(* Logix 5000 project; controller VET 1756-L62 rev 19.52; software revision 19.01; part 26 of 27 *)
(* tags used below, declared in another part *)
   _Sel_Comun : Selector;   // Comun selectores
   _Sel_eqp : Sel_eqp[300];   // Equipos Select
   _Sel_eqp_comun : Sel_eqp;   // Comun equqipos selector
   _Selector : Selector[80];
   Aux : DINT[40];
   Borrar : DINT[100];
   Color_aux : INT[1000];
   ecfgcom : Eqp_Cfg;
   eqpcom : Equipo;   // Comun Equipos
   OrigCom2 : Origen;
   SetDInt : DINT[500];
   Table1 : DINT[100];
   ti : Index;
   _BatCode : DINT[100];
   _Codes : DINT[500];
   _Eqp : Equipo[800];
   _Eqp_Cfg : Eqp_Cfg[800];
   _Origen : Origen[40];
   _Typlgie : Eqp_Typologie[800];   // Process Flow Typologie
   automat : DINT[100];
   comandos : DINT[10];
   DRT : DRTs[10];
   Set_Global : DINT[20];
   Tab_ODS : Tab_O_D_Orig;   // Tabla Origen Destino
(* Typlgie, continued *)

ROUTINE Main   (* ladder *)
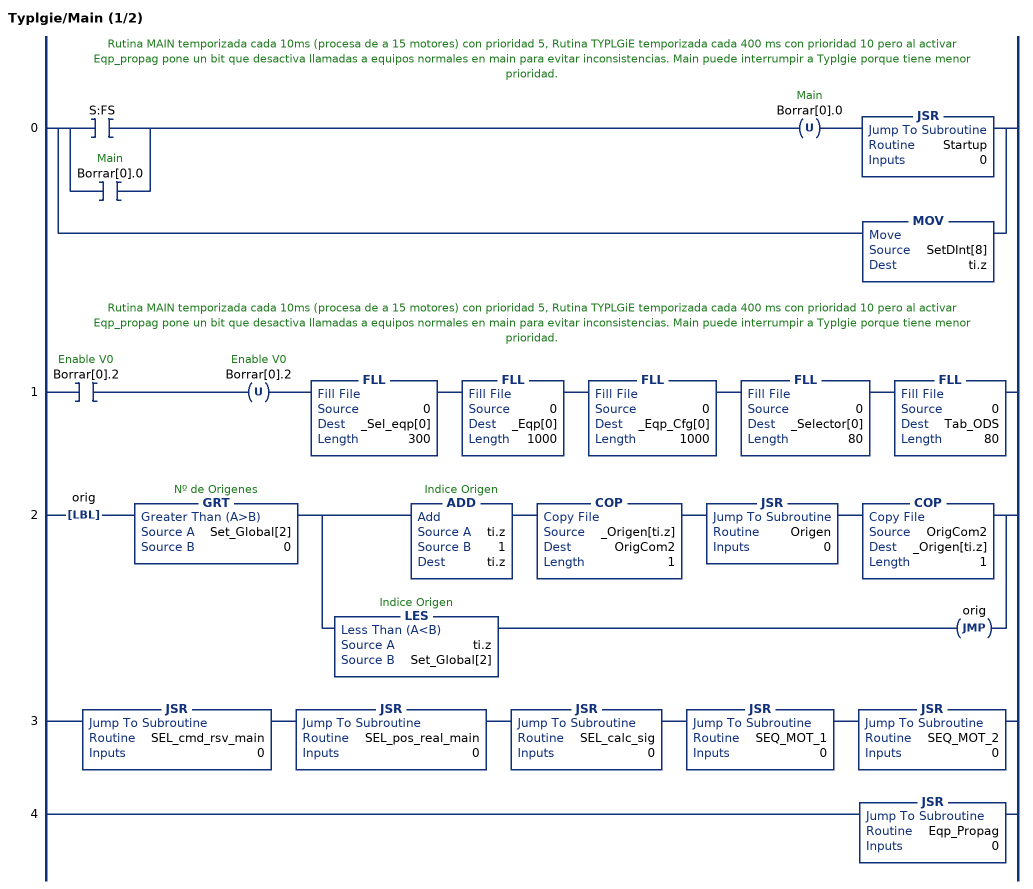
   // Rutina MAIN temporizada cada 10ms (procesa de a 15 motores) con prioridad 5, Rutina TYPLGiE temporizada cada 400 ms con prioridad 10 pero al activar Eqp_propag pone un bit que desactiva llamadas a equipos normales en main para evitar inconsistencias. Main puede interrumpir a Typlgie porque tiene menor prioridad.
   0: [[XIC(S:FS) ,XIC(Borrar[0].0) ] OTU(Borrar[0].0) JSR(Startup,0) ,MOV(SetDInt[8],ti.z) ];
   // Rutina MAIN temporizada cada 10ms (procesa de a 15 motores) con prioridad 5, Rutina TYPLGiE temporizada cada 400 ms con prioridad 10 pero al activar Eqp_propag pone un bit que desactiva llamadas a equipos normales en main para evitar inconsistencias. Main puede interrumpir a Typlgie porque tiene menor prioridad.
   1: XIC(Borrar[0].2)OTU(Borrar[0].2)FLL(0,_Sel_eqp[0],300)FLL(0,_Eqp[0],1000)FLL(0,_Eqp_Cfg[0],1000)FLL(0,_Selector[0],80)FLL(0,Tab_ODS,80);
   2: LBL(orig)GRT(Set_Global[2],0)[ADD(ti.z,1,ti.z) COP(_Origen[ti.z],OrigCom2,1) JSR(Origen,0) COP(OrigCom2,_Origen[ti.z],1) ,LES(ti.z,Set_Global[2]) JMP(orig) ];
   3: JSR(SEL_cmd_rsv_main,0)JSR(SEL_pos_real_main,0)JSR(SEL_calc_sig,0)JSR(SEQ_MOT_1,0)JSR(SEQ_MOT_2,0);
   4: JSR(Eqp_Propag,0);
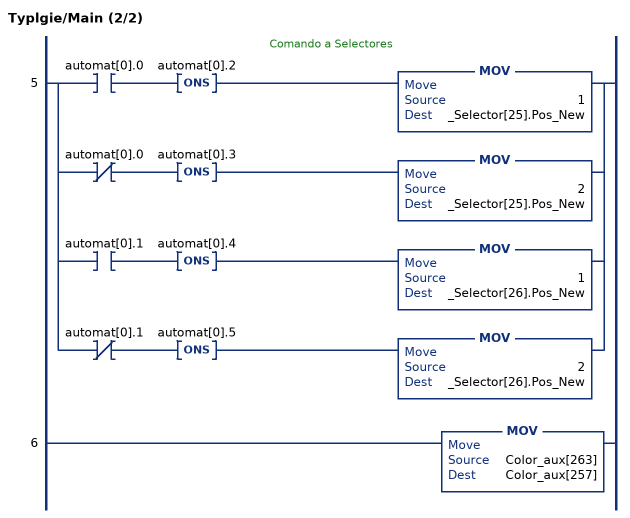
   // Comando a Selectores
   5: [[XIC(automat[0].0) ONS(automat[0].2) MOV(1,_Selector[25].Pos_New) ,XIO(automat[0].0) ONS(automat[0].3) MOV(2,_Selector[25].Pos_New) ] ,[XIC(automat[0].1) ONS(automat[0].4) MOV(1,_Selector[26].Pos_New) ,XIO(automat[0].1) ONS(automat[0].5) MOV(2,_Selector[26].Pos_New) ] ];
   6: MOV(Color_aux[263],Color_aux[257]);
END_ROUTINE

ROUTINE Origen   (* ladder *)
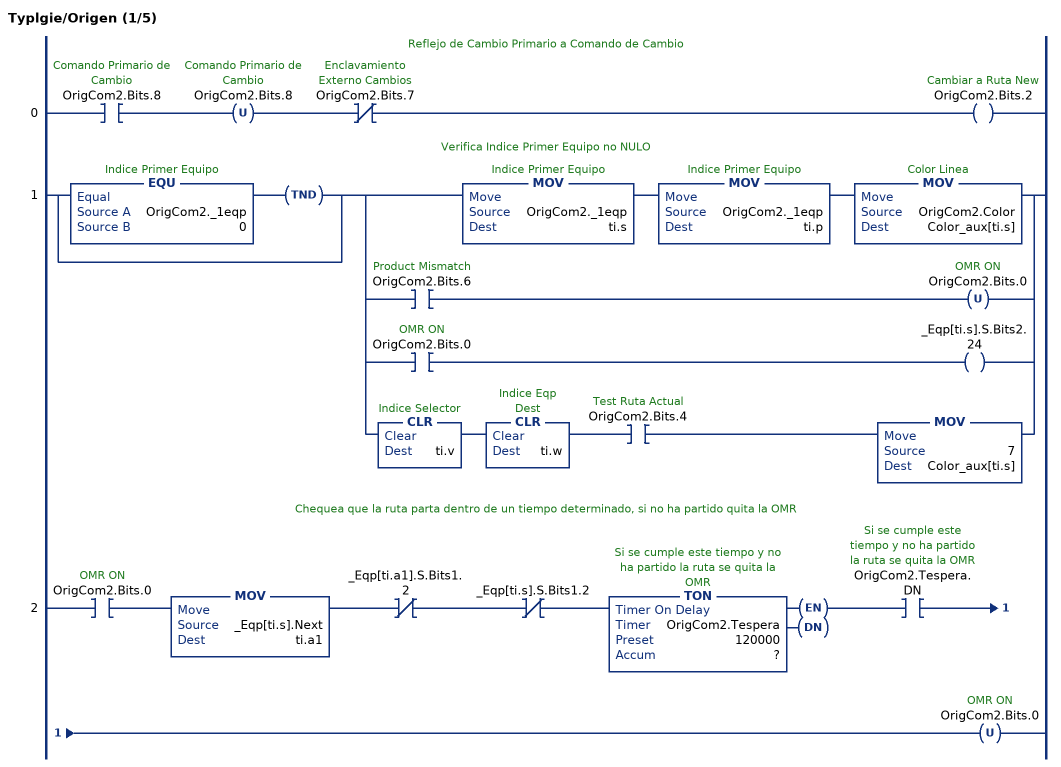
   // Reflejo de Cambio Primario a Comando de Cambio
   0: XIC(OrigCom2.Bits.8)OTU(OrigCom2.Bits.8)XIO(OrigCom2.Bits.7)OTE(OrigCom2.Bits.2);
   // Verifica Indice Primer Equipo no NULO
   1: [EQU(OrigCom2._1eqp,0) TND() ,][MOV(OrigCom2._1eqp,ti.s) MOV(OrigCom2._1eqp,ti.p) MOV(OrigCom2.Color,Color_aux[ti.s]) ,XIC(OrigCom2.Bits.6) OTU(OrigCom2.Bits.0) ,XIC(OrigCom2.Bits.0) OTE(_Eqp[ti.s].S.Bits2.24) ,CLR(ti.v) CLR(ti.w) XIC(OrigCom2.Bits.4) MOV(7,Color_aux[ti.s]) ];
   // Chequea que la ruta parta dentro de un tiempo determinado, si no ha partido quita la OMR
   2: XIC(OrigCom2.Bits.0)MOV(_Eqp[ti.s].Next,ti.a1)XIO(_Eqp[ti.a1].S.Bits1.2)XIO(_Eqp[ti.s].S.Bits1.2)TON(OrigCom2.Tespera,?,?)XIC(OrigCom2.Tespera.DN)OTU(OrigCom2.Bits.0);
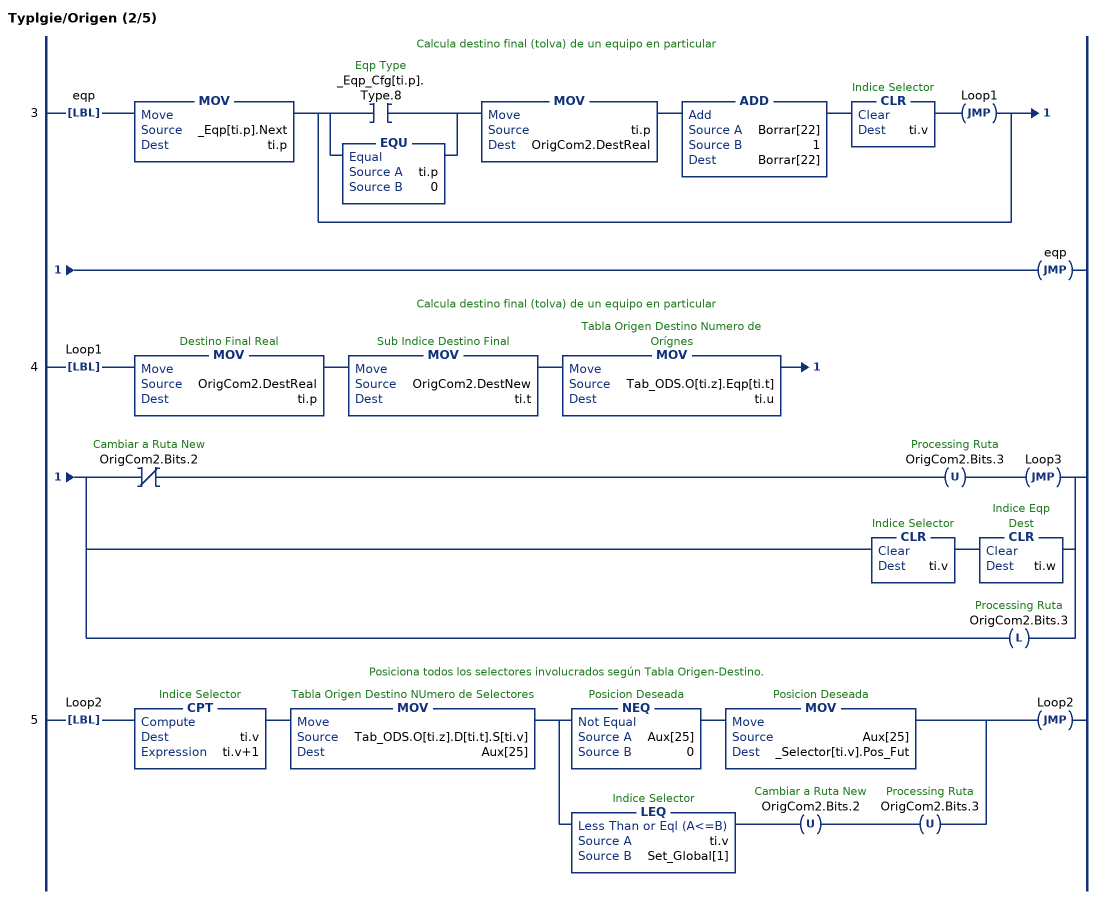
   // Calcula destino final (tolva) de un equipo en particular
   3: LBL(eqp)MOV(_Eqp[ti.p].Next,ti.p)[[XIC(_Eqp_Cfg[ti.p].Type.8) ,EQU(ti.p,0) ] MOV(ti.p,OrigCom2.DestReal) ADD(Borrar[22],1,Borrar[22]) CLR(ti.v) JMP(Loop1) ,]JMP(eqp);
   // Calcula destino final (tolva) de un equipo en particular
   4: LBL(Loop1)MOV(OrigCom2.DestReal,ti.p)MOV(OrigCom2.DestNew,ti.t)MOV(Tab_ODS.O[ti.z].Eqp[ti.t],ti.u)[XIO(OrigCom2.Bits.2) OTU(OrigCom2.Bits.3) JMP(Loop3) ,CLR(ti.v) CLR(ti.w) ,OTL(OrigCom2.Bits.3) ];
   // Posiciona todos los selectores involucrados según Tabla Origen-Destino.
   5: LBL(Loop2)CPT(ti.v,ti.v+1)MOV(Tab_ODS.O[ti.z].D[ti.t].S[ti.v],Aux[25])[NEQ(Aux[25],0) MOV(Aux[25],_Selector[ti.v].Pos_Fut) ,LEQ(ti.v,Set_Global[1]) OTU(OrigCom2.Bits.2) OTU(OrigCom2.Bits.3) ]JMP(Loop2);
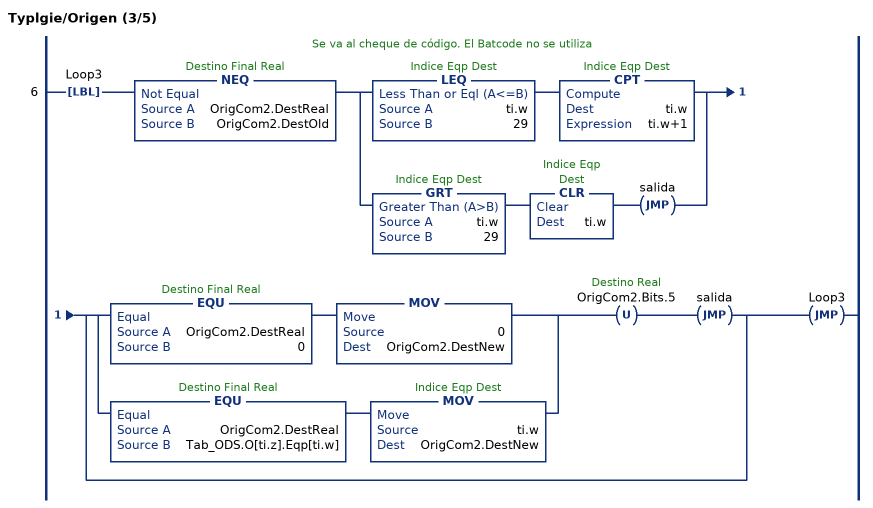
   // Se va al cheque de código. El Batcode no se utiliza
   6: LBL(Loop3)NEQ(OrigCom2.DestReal,OrigCom2.DestOld)[LEQ(ti.w,29) CPT(ti.w,ti.w+1) ,GRT(ti.w,29) CLR(ti.w) JMP(salida) ][[EQU(OrigCom2.DestReal,0) MOV(0,OrigCom2.DestNew) ,EQU(OrigCom2.DestReal,Tab_ODS.O[ti.z].Eqp[ti.w]) MOV(ti.w,OrigCom2.DestNew) ] OTU(OrigCom2.Bits.5) JMP(salida) ,]JMP(Loop3);
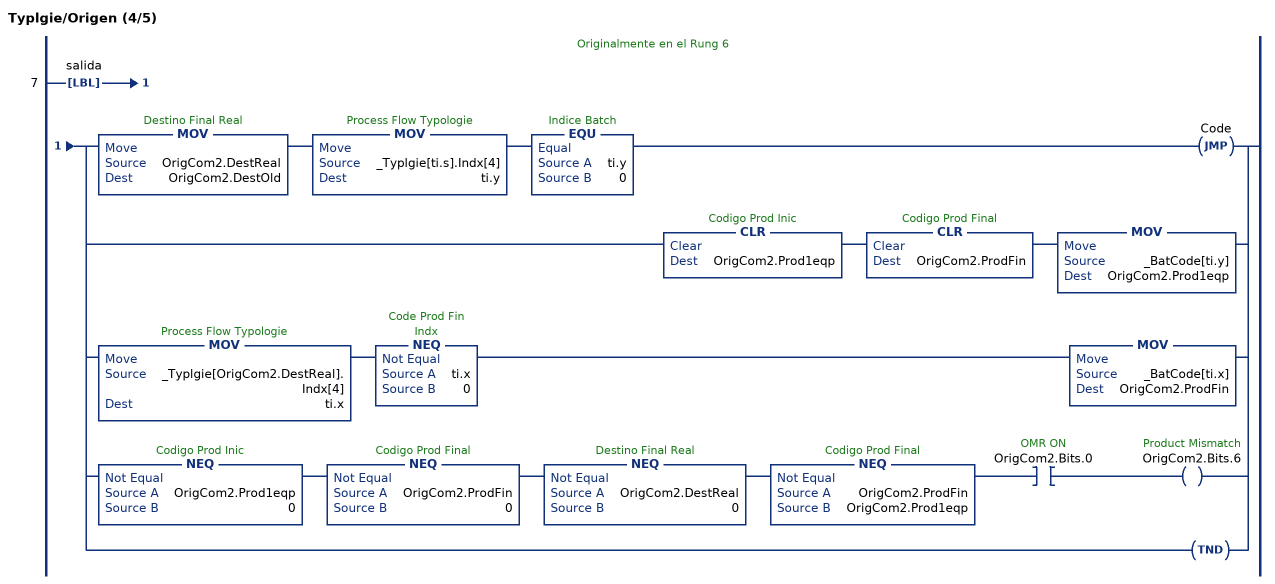
   // Originalmente en el Rung 6
   7: LBL(salida)[MOV(OrigCom2.DestReal,OrigCom2.DestOld) MOV(_Typlgie[ti.s].Indx[4],ti.y) EQU(ti.y,0) JMP(Code) ,CLR(OrigCom2.Prod1eqp) CLR(OrigCom2.ProdFin) MOV(_BatCode[ti.y],OrigCom2.Prod1eqp) ,MOV(_Typlgie[OrigCom2.DestReal].Indx[4],ti.x) NEQ(ti.x,0) MOV(_BatCode[ti.x],OrigCom2.ProdFin) ,NEQ(OrigCom2.Prod1eqp,0) NEQ(OrigCom2.ProdFin,0) NEQ(OrigCom2.DestReal,0) NEQ(OrigCom2.ProdFin,OrigCom2.Prod1eqp) XIC(OrigCom2.Bits.0) OTE(OrigCom2.Bits.6) ,TND() ];
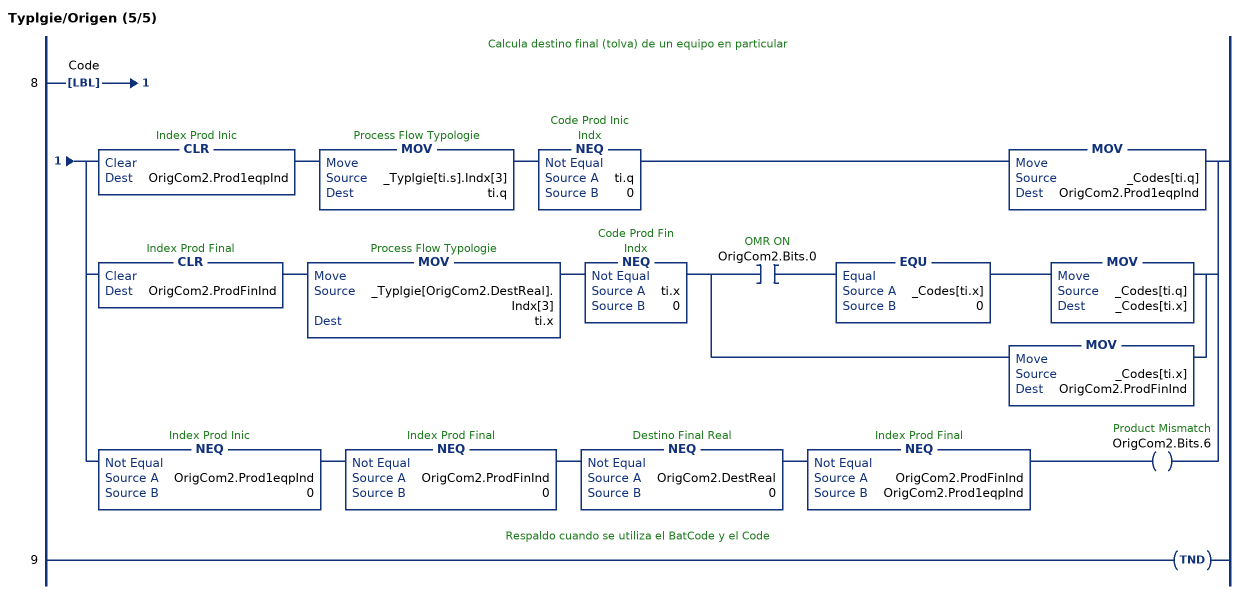
   // Calcula destino final (tolva) de un equipo en particular
   8: LBL(Code)[CLR(OrigCom2.Prod1eqpInd) MOV(_Typlgie[ti.s].Indx[3],ti.q) NEQ(ti.q,0) MOV(_Codes[ti.q],OrigCom2.Prod1eqpInd) ,CLR(OrigCom2.ProdFinInd) MOV(_Typlgie[OrigCom2.DestReal].Indx[3],ti.x) NEQ(ti.x,0) [XIC(OrigCom2.Bits.0) EQU(_Codes[ti.x],0) MOV(_Codes[ti.q],_Codes[ti.x]) ,MOV(_Codes[ti.x],OrigCom2.ProdFinInd) ] ,NEQ(OrigCom2.Prod1eqpInd,0) NEQ(OrigCom2.ProdFinInd,0) NEQ(OrigCom2.DestReal,0) NEQ(OrigCom2.ProdFinInd,OrigCom2.Prod1eqpInd) OTE(OrigCom2.Bits.6) ];
   // Respaldo cuando se utiliza el BatCode y el Code
   9: TND();
END_ROUTINE

ROUTINE SEL_calc_sig   (* ladder *)
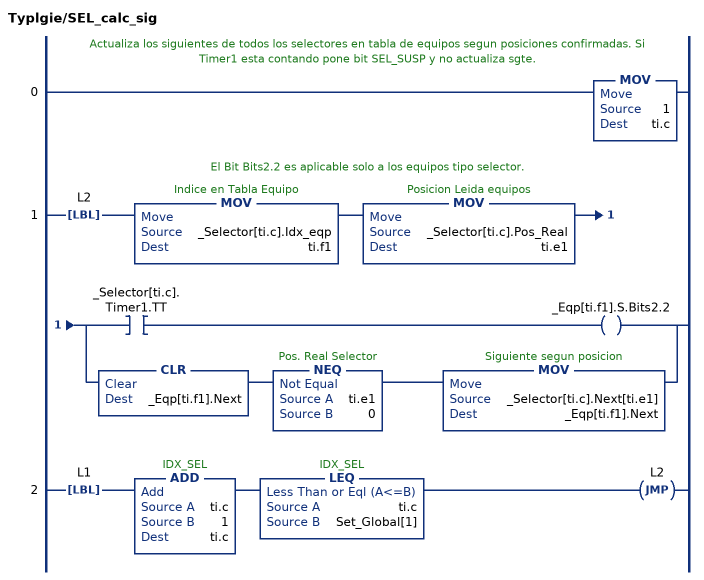
   // Actualiza los siguientes de todos los selectores en tabla de equipos segun posiciones confirmadas. Si Timer1 esta contando pone bit SEL_SUSP y no actualiza sgte.
   0: MOV(1,ti.c);
   // El Bit Bits2.2 es aplicable solo a los equipos tipo selector.
   1: LBL(L2)MOV(_Selector[ti.c].Idx_eqp,ti.f1)MOV(_Selector[ti.c].Pos_Real,ti.e1)[XIC(_Selector[ti.c].Timer1.TT) OTE(_Eqp[ti.f1].S.Bits2.2) ,CLR(_Eqp[ti.f1].Next) NEQ(ti.e1,0) MOV(_Selector[ti.c].Next[ti.e1],_Eqp[ti.f1].Next) ];
   2: LBL(L1)ADD(ti.c,1,ti.c)LEQ(ti.c,Set_Global[1])JMP(L2);
END_ROUTINE

ROUTINE SEL_cmd_rsv   (* ladder *)
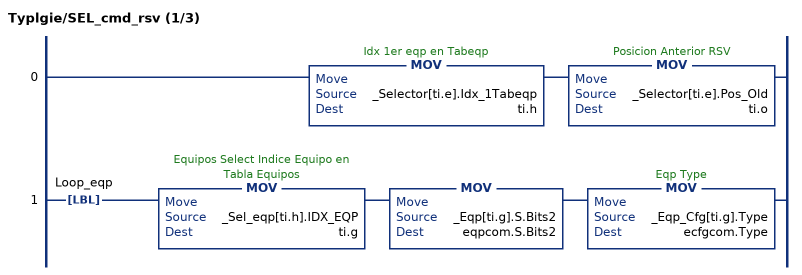
   0: MOV(_Selector[ti.e].Idx_1Tabeqp,ti.h)MOV(_Selector[ti.e].Pos_Old,ti.o);
   1: LBL(Loop_eqp)MOV(_Sel_eqp[ti.h].IDX_EQP,ti.g)MOV(_Eqp[ti.g].S.Bits2,eqpcom.S.Bits2)MOV(_Eqp_Cfg[ti.g].Type,ecfgcom.Type);
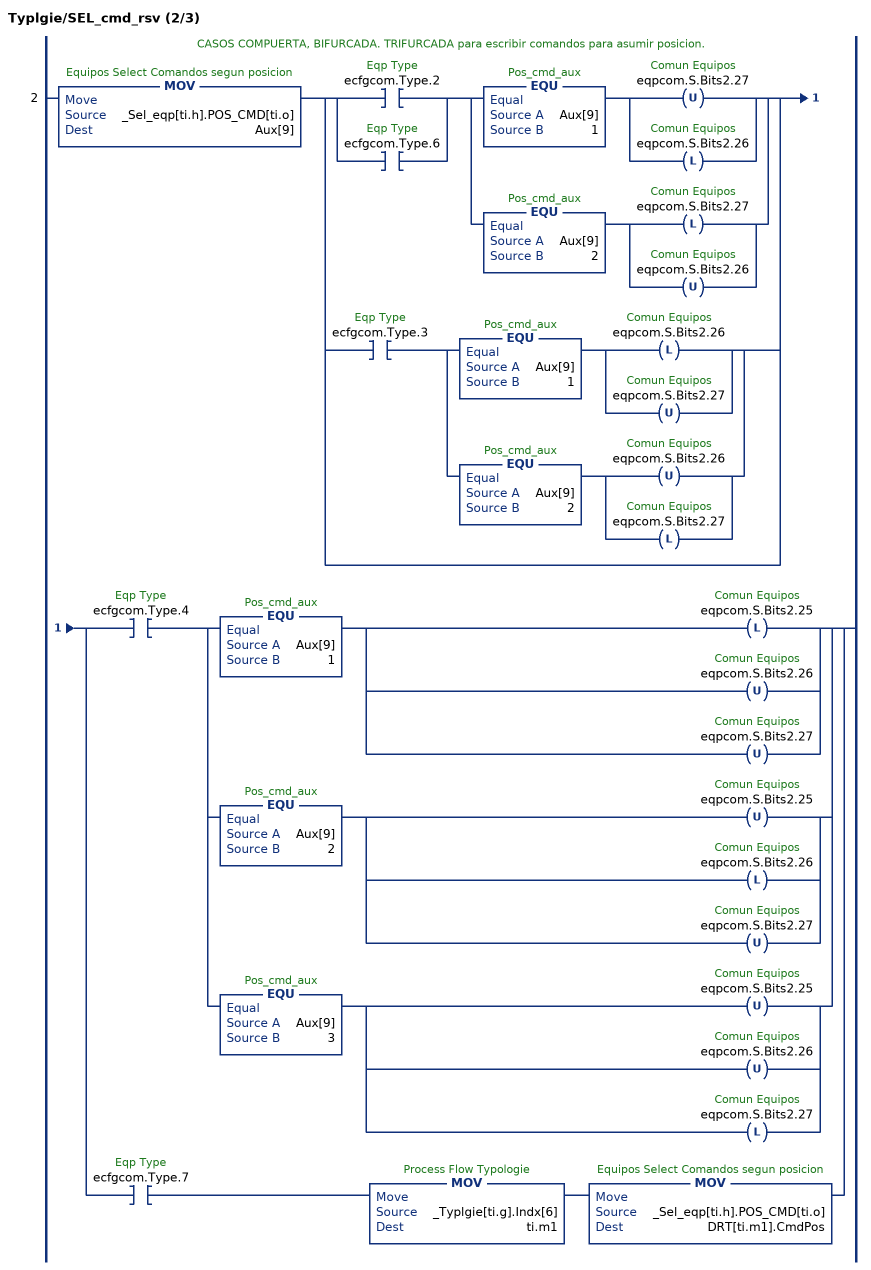
   // CASOS COMPUERTA, BIFURCADA. TRIFURCADA para escribir comandos para asumir posicion.
   2: MOV(_Sel_eqp[ti.h].POS_CMD[ti.o],Aux[9])[[XIC(ecfgcom.Type.2) ,XIC(ecfgcom.Type.6) ] [EQU(Aux[9],1) [OTU(eqpcom.S.Bits2.27) ,OTL(eqpcom.S.Bits2.26) ] ,EQU(Aux[9],2) [OTL(eqpcom.S.Bits2.27) ,OTU(eqpcom.S.Bits2.26) ] ] ,XIC(ecfgcom.Type.3) [EQU(Aux[9],1) [OTL(eqpcom.S.Bits2.26) ,OTU(eqpcom.S.Bits2.27) ] ,EQU(Aux[9],2) [OTU(eqpcom.S.Bits2.26) ,OTL(eqpcom.S.Bits2.27) ] ] ,][XIC(ecfgcom.Type.4) [EQU(Aux[9],1) [OTL(eqpcom.S.Bits2.25) ,OTU(eqpcom.S.Bits2.26) ,OTU(eqpcom.S.Bits2.27) ] ,EQU(Aux[9],2) [OTU(eqpcom.S.Bits2.25) ,OTL(eqpcom.S.Bits2.26) ,OTU(eqpcom.S.Bits2.27) ] ,EQU(Aux[9],3) [OTU(eqpcom.S.Bits2.25) ,OTU(eqpcom.S.Bits2.26) ,OTL(eqpcom.S.Bits2.27) ] ] ,XIC(ecfgcom.Type.7) MOV(_Typlgie[ti.g].Indx[6],ti.m1) MOV(_Sel_eqp[ti.h].POS_CMD[ti.o],DRT[ti.m1].CmdPos) ];
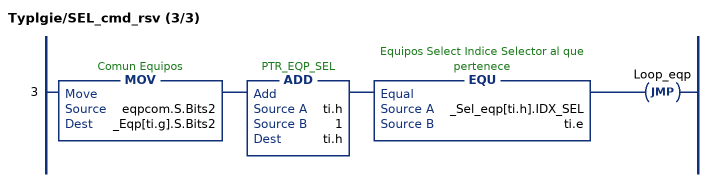
   3: MOV(eqpcom.S.Bits2,_Eqp[ti.g].S.Bits2)ADD(ti.h,1,ti.h)EQU(_Sel_eqp[ti.h].IDX_SEL,ti.e)JMP(Loop_eqp);
END_ROUTINE

ROUTINE SEL_cmd_rsv_main   (* ladder *)
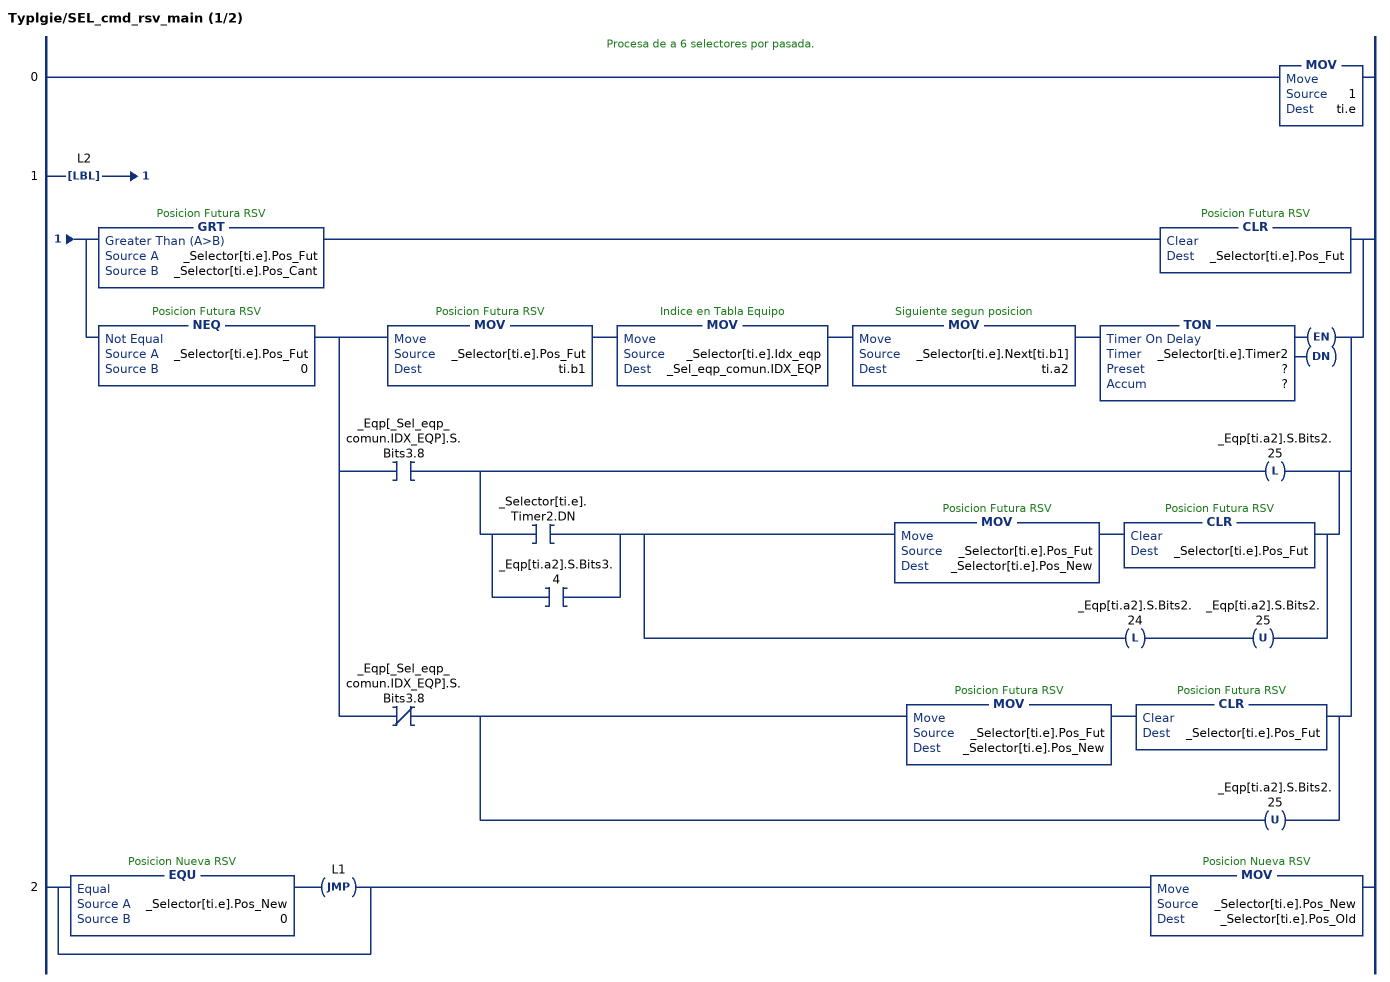
   // Procesa de a 6 selectores por pasada.
   0: MOV(1,ti.e);
   1: LBL(L2)[GRT(_Selector[ti.e].Pos_Fut,_Selector[ti.e].Pos_Cant) CLR(_Selector[ti.e].Pos_Fut) ,NEQ(_Selector[ti.e].Pos_Fut,0) [MOV(_Selector[ti.e].Pos_Fut,ti.b1) MOV(_Selector[ti.e].Idx_eqp,_Sel_eqp_comun.IDX_EQP) MOV(_Selector[ti.e].Next[ti.b1],ti.a2) TON(_Selector[ti.e].Timer2,?,?) ,XIC(_Eqp[_Sel_eqp_comun.IDX_EQP].S.Bits3.8) [OTL(_Eqp[ti.a2].S.Bits2.25) ,[XIC(_Selector[ti.e].Timer2.DN) ,XIC(_Eqp[ti.a2].S.Bits3.4) ] [MOV(_Selector[ti.e].Pos_Fut,_Selector[ti.e].Pos_New) CLR(_Selector[ti.e].Pos_Fut) ,OTL(_Eqp[ti.a2].S.Bits2.24) OTU(_Eqp[ti.a2].S.Bits2.25) ] ] ,XIO(_Eqp[_Sel_eqp_comun.IDX_EQP].S.Bits3.8) [MOV(_Selector[ti.e].Pos_Fut,_Selector[ti.e].Pos_New) CLR(_Selector[ti.e].Pos_Fut) ,OTU(_Eqp[ti.a2].S.Bits2.25) ] ] ];
   2: [EQU(_Selector[ti.e].Pos_New,0) JMP(L1) ,]MOV(_Selector[ti.e].Pos_New,_Selector[ti.e].Pos_Old);
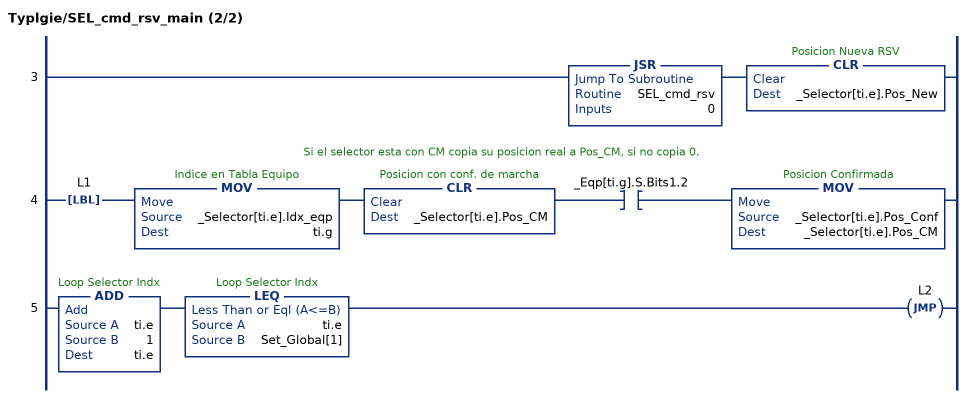
   3: JSR(SEL_cmd_rsv,0)CLR(_Selector[ti.e].Pos_New);
   // Si el selector esta con CM copia su posicion real a Pos_CM, si no copia 0.
   4: LBL(L1)MOV(_Selector[ti.e].Idx_eqp,ti.g)CLR(_Selector[ti.e].Pos_CM)XIC(_Eqp[ti.g].S.Bits1.2)MOV(_Selector[ti.e].Pos_Conf,_Selector[ti.e].Pos_CM);
   5: ADD(ti.e,1,ti.e)LEQ(ti.e,Set_Global[1])JMP(L2);
END_ROUTINE

ROUTINE SEL_pos_real   (* ladder *)
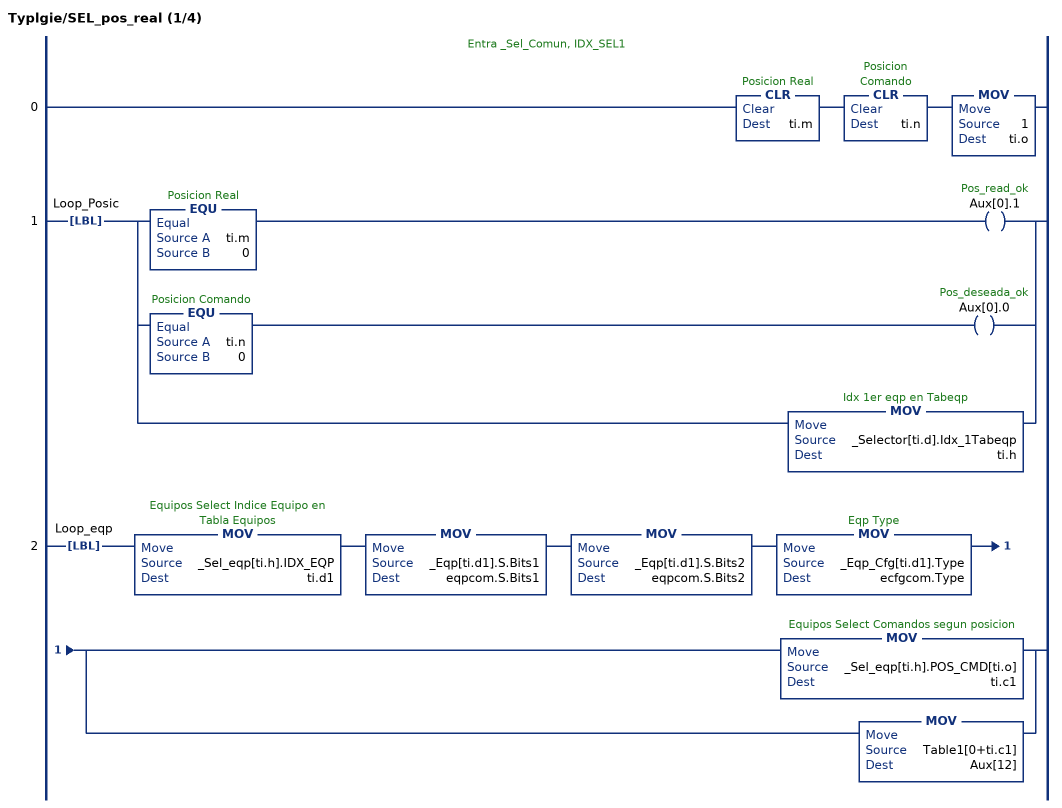
   // Entra _Sel_Comun, IDX_SEL1
   0: CLR(ti.m)CLR(ti.n)MOV(1,ti.o);
   1: LBL(Loop_Posic)[EQU(ti.m,0) OTE(Aux[0].1) ,EQU(ti.n,0) OTE(Aux[0].0) ,MOV(_Selector[ti.d].Idx_1Tabeqp,ti.h) ];
   2: LBL(Loop_eqp)MOV(_Sel_eqp[ti.h].IDX_EQP,ti.d1)MOV(_Eqp[ti.d1].S.Bits1,eqpcom.S.Bits1)MOV(_Eqp[ti.d1].S.Bits2,eqpcom.S.Bits2)MOV(_Eqp_Cfg[ti.d1].Type,ecfgcom.Type)[MOV(_Sel_eqp[ti.h].POS_CMD[ti.o],ti.c1) ,MOV(Table1[0+ti.c1],Aux[12]) ];
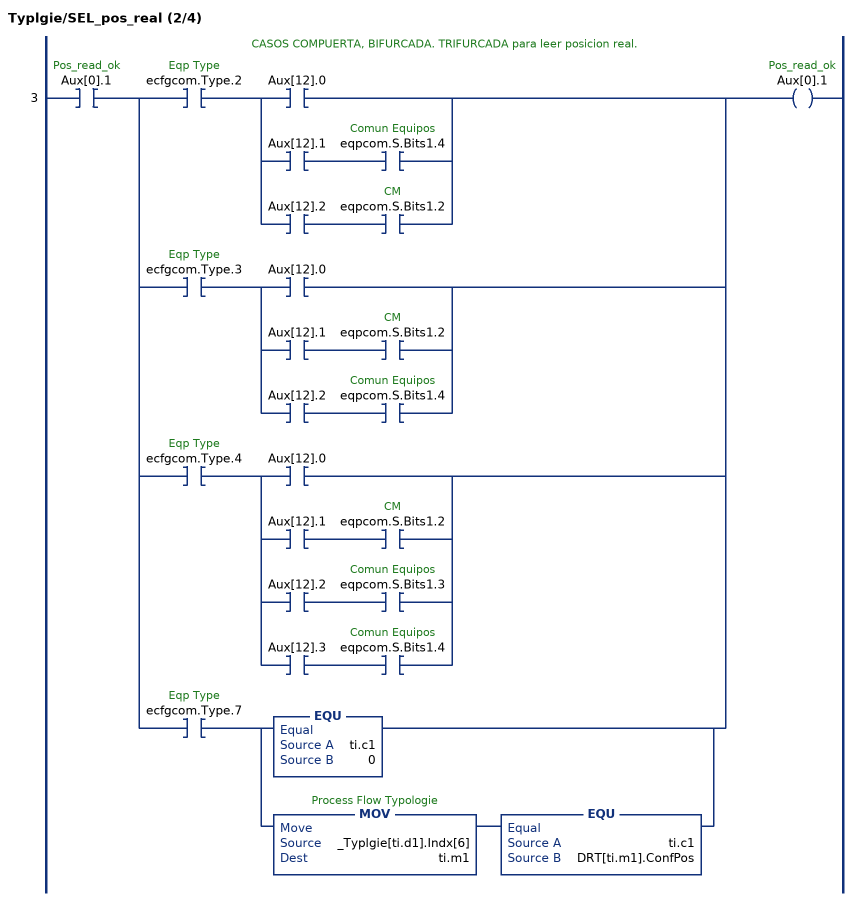
   // CASOS COMPUERTA, BIFURCADA. TRIFURCADA para leer posicion real.
   3: XIC(Aux[0].1)[XIC(ecfgcom.Type.2) [XIC(Aux[12].0) ,XIC(Aux[12].1) XIC(eqpcom.S.Bits1.4) ,XIC(Aux[12].2) XIC(eqpcom.S.Bits1.2) ] ,XIC(ecfgcom.Type.3) [XIC(Aux[12].0) ,XIC(Aux[12].1) XIC(eqpcom.S.Bits1.2) ,XIC(Aux[12].2) XIC(eqpcom.S.Bits1.4) ] ,XIC(ecfgcom.Type.4) [XIC(Aux[12].0) ,XIC(Aux[12].1) XIC(eqpcom.S.Bits1.2) ,XIC(Aux[12].2) XIC(eqpcom.S.Bits1.3) ,XIC(Aux[12].3) XIC(eqpcom.S.Bits1.4) ] ,XIC(ecfgcom.Type.7) [EQU(ti.c1,0) ,MOV(_Typlgie[ti.d1].Indx[6],ti.m1) EQU(ti.c1,DRT[ti.m1].ConfPos) ] ]OTE(Aux[0].1);
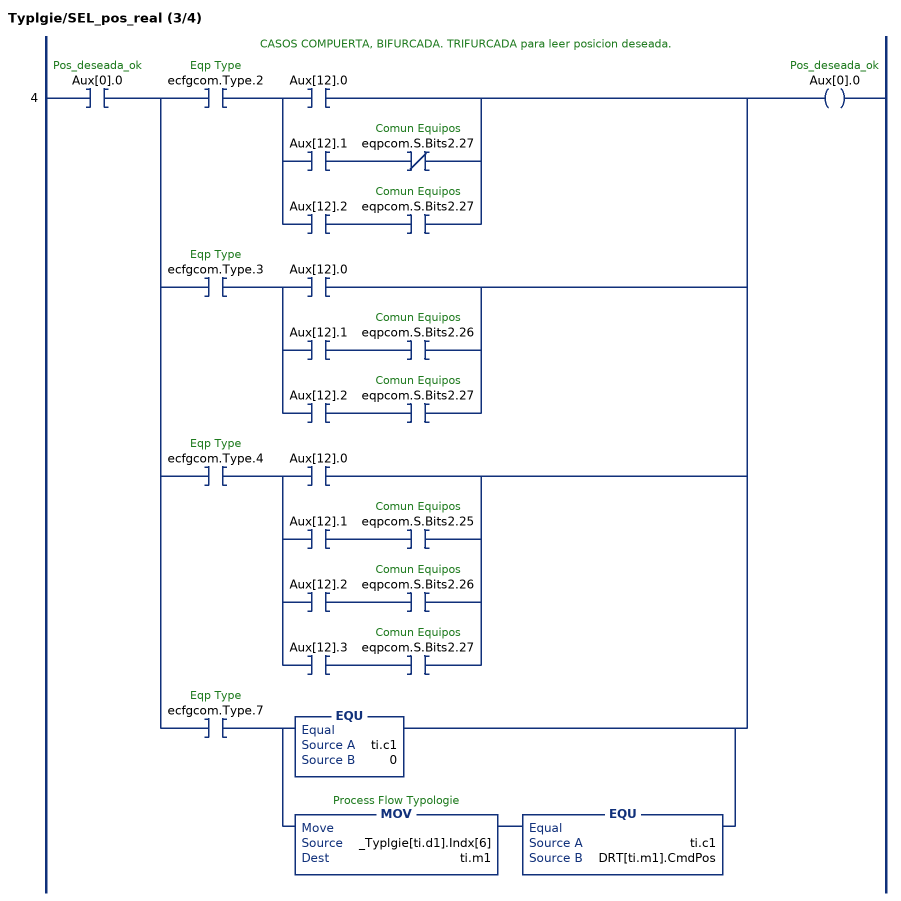
   // CASOS COMPUERTA, BIFURCADA. TRIFURCADA para leer posicion deseada.
   4: XIC(Aux[0].0)[XIC(ecfgcom.Type.2) [XIC(Aux[12].0) ,XIC(Aux[12].1) XIO(eqpcom.S.Bits2.27) ,XIC(Aux[12].2) XIC(eqpcom.S.Bits2.27) ] ,XIC(ecfgcom.Type.3) [XIC(Aux[12].0) ,XIC(Aux[12].1) XIC(eqpcom.S.Bits2.26) ,XIC(Aux[12].2) XIC(eqpcom.S.Bits2.27) ] ,XIC(ecfgcom.Type.4) [XIC(Aux[12].0) ,XIC(Aux[12].1) XIC(eqpcom.S.Bits2.25) ,XIC(Aux[12].2) XIC(eqpcom.S.Bits2.26) ,XIC(Aux[12].3) XIC(eqpcom.S.Bits2.27) ] ,XIC(ecfgcom.Type.7) [EQU(ti.c1,0) ,MOV(_Typlgie[ti.d1].Indx[6],ti.m1) EQU(ti.c1,DRT[ti.m1].CmdPos) ] ]OTE(Aux[0].0);
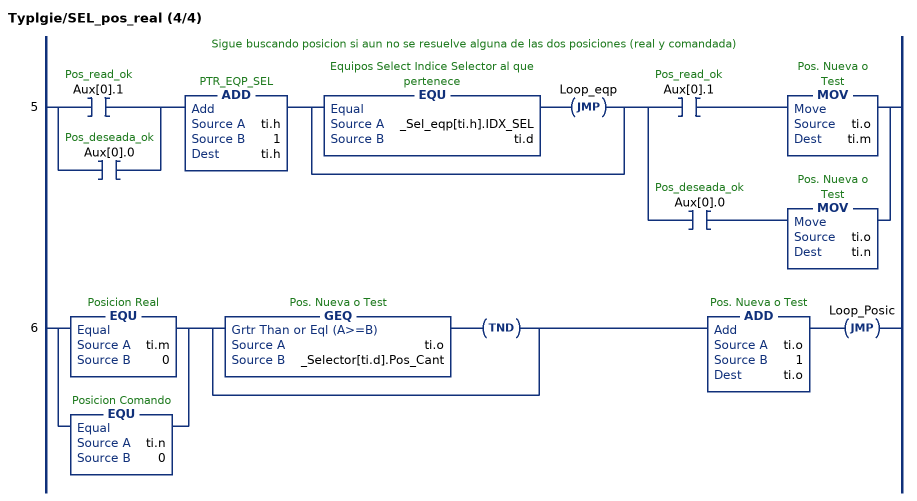
   // Sigue buscando posicion si aun no se resuelve alguna de las dos posiciones (real y comandada)
   5: [XIC(Aux[0].1) ,XIC(Aux[0].0) ]ADD(ti.h,1,ti.h)[EQU(_Sel_eqp[ti.h].IDX_SEL,ti.d) JMP(Loop_eqp) ,][XIC(Aux[0].1) MOV(ti.o,ti.m) ,XIC(Aux[0].0) MOV(ti.o,ti.n) ];
   6: [EQU(ti.m,0) ,EQU(ti.n,0) ][GEQ(ti.o,_Selector[ti.d].Pos_Cant) TND() ,]ADD(ti.o,1,ti.o)JMP(Loop_Posic);
END_ROUTINE

ROUTINE SEL_pos_real_main   (* ladder *)
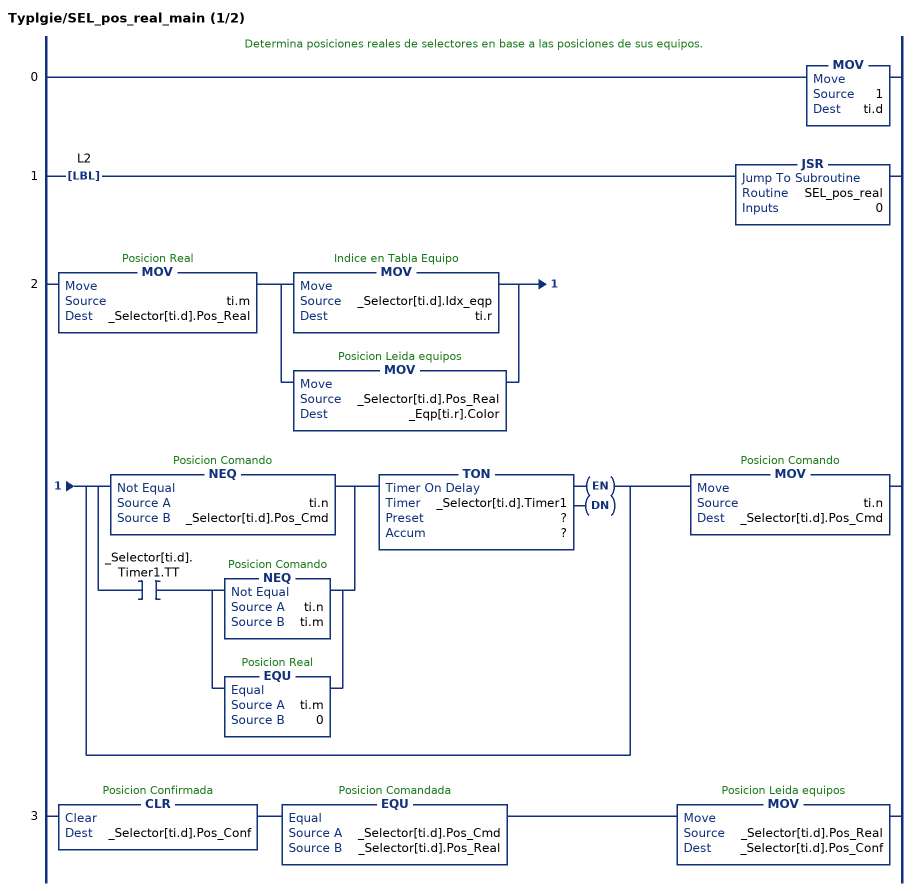
   // Determina posiciones reales de selectores en base a las posiciones de sus equipos.
   0: MOV(1,ti.d);
   1: LBL(L2)JSR(SEL_pos_real,0);
   2: MOV(ti.m,_Selector[ti.d].Pos_Real)[MOV(_Selector[ti.d].Idx_eqp,ti.r) ,MOV(_Selector[ti.d].Pos_Real,_Eqp[ti.r].Color) ][[NEQ(ti.n,_Selector[ti.d].Pos_Cmd) ,XIC(_Selector[ti.d].Timer1.TT) [NEQ(ti.n,ti.m) ,EQU(ti.m,0) ] ] TON(_Selector[ti.d].Timer1,?,?) ,]MOV(ti.n,_Selector[ti.d].Pos_Cmd);
   3: CLR(_Selector[ti.d].Pos_Conf)EQU(_Selector[ti.d].Pos_Cmd,_Selector[ti.d].Pos_Real)MOV(_Selector[ti.d].Pos_Real,_Selector[ti.d].Pos_Conf);
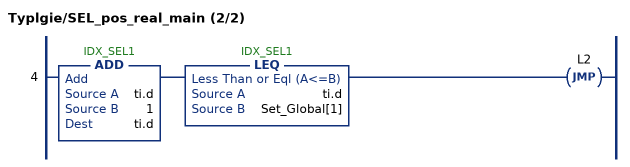
   4: ADD(ti.d,1,ti.d)LEQ(ti.d,Set_Global[1])JMP(L2);
END_ROUTINE
